(* PLC project Sin nombre, Desconocido Sin nombre 1 *)
(* stored: creationDateTime 2022-11-05T08:40:31, modificationDateTime 2022-11-06T14:33:46 *)

PROGRAM prueba
  VAR
    sensor_hall AT %IX0.0 : BOOL := 0;
    led AT %QX0.0 : BOOL := 1;
    led_rojo AT %QX0.2 : BOOL := 0;
    rele AT %QX0.1 : BOOL := 0;
  END_VAR
  VAR
    subir_pist : TP;
    counter : CTU;
    delay : TON;
    bajar_pist : TP;
  END_VAR
  VAR  (* added by the conversion: wires and edge detectors of the diagram *)
    R_TRIG1 : R_TRIG;
    _NOT16_OUT : BOOL;
  END_VAR

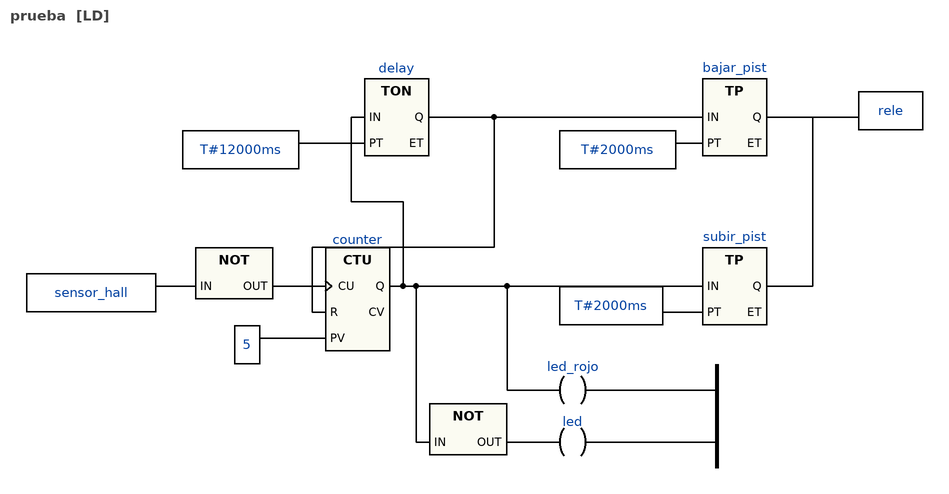
(* LD diagram, written out as Structured Text *)
R_TRIG1(CLK := NOT sensor_hall);
delay(IN := counter.Q, PT := T#12000ms);
counter(CU := R_TRIG1.Q, R := delay.Q, PV := 5);
subir_pist(IN := counter.Q, PT := T#2000ms);
bajar_pist(IN := delay.Q, PT := T#2000ms);
rele := subir_pist.Q OR bajar_pist.Q;
led_rojo := counter.Q;
_NOT16_OUT := NOT counter.Q;
led := _NOT16_OUT;
END_PROGRAM

CONFIGURATION Config0
  RESOURCE Res0 ON PLC
    TASK task0(INTERVAL := T#20ms, PRIORITY := 0);
    PROGRAM instance0 WITH task0 : prueba;
  END_RESOURCE
END_CONFIGURATION
